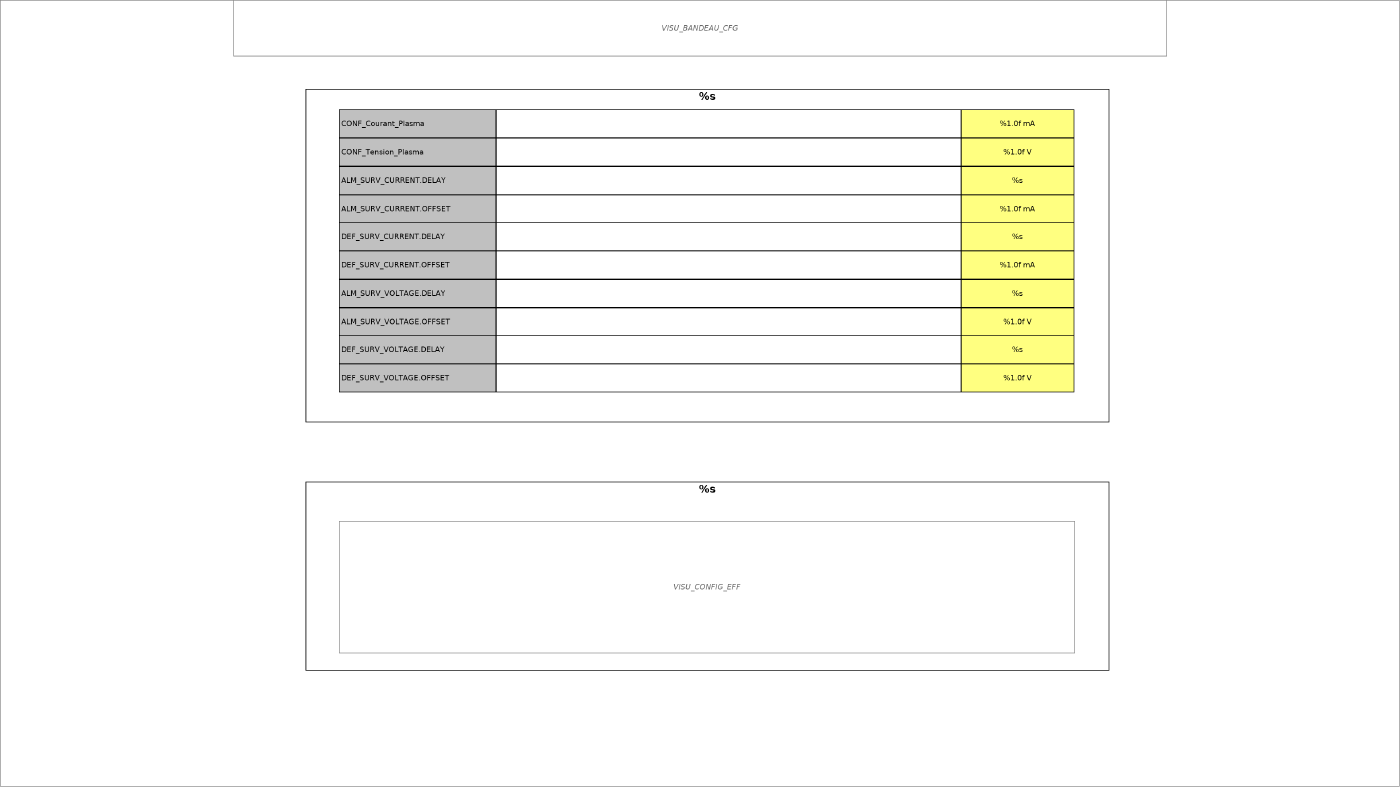
VISUALIZATION VISU_CONFIG_EFFLUV  // 1920x1080, background image fond_blanc_1280_1024
    Frame (320,0 1280x77)
        shows VISU_BANDEAU_CFG()
    RoundedRectangle (419,122 1102x457), "%s", text list: 'TextList_Config_EFFLUVAGE', text index: 0
    Rectangle (465,150 215x39), "CONF_Courant_Plasma"
    Rectangle (680,150 638x39), text list: 'TextList_Config_EFFLUVAGE', text index: 8
    Rectangle (1318,150 155x39), "%1.0f mA", text variable: PRG_EFFLUVAGE.Effluvage.ALEFF.CONF_Courant_Plasma, input disabled if: NOT Global_Variables.PRG_USER.ACTU_USER.CONF_MACHINE
        OnMouseClick: write the text variable via InputWithLimits, min 0, max 100
    Rectangle (465,189 215x39), "CONF_Tension_Plasma"
    Rectangle (680,189 638x39), text list: 'TextList_Config_EFFLUVAGE', text index: 9
    Rectangle (1318,189 155x39), "%1.0f V", text variable: PRG_EFFLUVAGE.Effluvage.ALEFF.CONF_Tension_Plasma, input disabled if: NOT Global_Variables.PRG_USER.ACTU_USER.CONF_MACHINE
        OnMouseClick: write the text variable via InputWithLimits, min 0, max 100
    Rectangle (465,228 215x39), "ALM_SURV_CURRENT.DELAY"
    Rectangle (680,228 638x39), text list: 'TextList_Config_EFFLUVAGE', text index: 11
    Rectangle (1318,228 155x39), "%s", text variable: PRG_EFFLUVAGE.Effluvage.ALEFF.ALM_Surv_Current.DELAY, input disabled if: NOT Global_Variables.PRG_USER.ACTU_USER.CONF_MACHINE
        OnMouseClick: write the text variable via InputWithLimits, min 0
    Rectangle (465,267 215x39), "ALM_SURV_CURRENT.OFFSET"
    Rectangle (680,267 638x39), text list: 'TextList_Config_EFFLUVAGE', text index: 12
    Rectangle (1318,267 155x39), "%1.0f mA", text variable: PRG_EFFLUVAGE.Effluvage.ALEFF.VAR_ALM_SURV_CURRENT.OFFSET, input disabled if: NOT Global_Variables.PRG_USER.ACTU_USER.CONF_MACHINE
        OnMouseClick: write the text variable via InputWithLimits, min 0, max 100
    Rectangle (465,305 215x39), "DEF_SURV_CURRENT.DELAY"
    Rectangle (680,305 638x39), text list: 'TextList_Config_EFFLUVAGE', text index: 13
    Rectangle (1318,305 155x39), "%s", text variable: PRG_EFFLUVAGE.Effluvage.ALEFF.DEF_Surv_Current.DELAY, input disabled if: NOT Global_Variables.PRG_USER.ACTU_USER.CONF_MACHINE
        OnMouseClick: write the text variable via InputWithLimits, min 0
    Rectangle (465,344 215x39), "DEF_SURV_CURRENT.OFFSET"
    Rectangle (680,344 638x39), text list: 'TextList_Config_EFFLUVAGE', text index: 14
    Rectangle (1318,344 155x39), "%1.0f mA", text variable: PRG_EFFLUVAGE.Effluvage.ALEFF.VAR_DEF_SURV_CURRENT.OFFSET, input disabled if: NOT Global_Variables.PRG_USER.ACTU_USER.CONF_MACHINE
        OnMouseClick: write the text variable via InputWithLimits, min 0, max 100
    RoundedRectangle (419,661 1102x259), "%s", text list: 'TextList_Config_EFFLUVAGE', text index: 0
    Frame (465,715 1009x181)
        shows VISU_CONFIG_EFF(m_Input_PRG_EFFLUVAGE := PRG_EFFLUVAGE)
    Rectangle (465,383 215x39), "ALM_SURV_VOLTAGE.DELAY"
    Rectangle (680,383 638x39), text list: 'TextList_Config_EFFLUVAGE', text index: 11
    Rectangle (1318,383 155x39), "%s", text variable: PRG_EFFLUVAGE.Effluvage.ALEFF.ALM_Surv_Voltage.DELAY, input disabled if: NOT Global_Variables.PRG_USER.ACTU_USER.CONF_MACHINE
        OnMouseClick: write the text variable via InputWithLimits, min 0
    Rectangle (465,422 215x39), "ALM_SURV_VOLTAGE.OFFSET"
    Rectangle (680,422 638x39), text list: 'TextList_Config_EFFLUVAGE', text index: 12
    Rectangle (1318,422 155x39), "%1.0f V", text variable: PRG_EFFLUVAGE.Effluvage.ALEFF.VAR_ALM_SURV_VOLTAGE.OFFSET, input disabled if: NOT Global_Variables.PRG_USER.ACTU_USER.CONF_MACHINE
        OnMouseClick: write the text variable via InputWithLimits, min 0, max 100
    Rectangle (465,460 215x39), "DEF_SURV_VOLTAGE.DELAY"
    Rectangle (680,460 638x39), text list: 'TextList_Config_EFFLUVAGE', text index: 13
    Rectangle (1318,460 155x39), "%s", text variable: PRG_EFFLUVAGE.Effluvage.ALEFF.DEF_Surv_Voltage.DELAY, input disabled if: NOT Global_Variables.PRG_USER.ACTU_USER.CONF_MACHINE
        OnMouseClick: write the text variable via InputWithLimits, min 0
    Rectangle (465,499 215x39), "DEF_SURV_VOLTAGE.OFFSET"
    Rectangle (680,499 638x39), text list: 'TextList_Config_EFFLUVAGE', text index: 14
    Rectangle (1318,499 155x39), "%1.0f V", text variable: PRG_EFFLUVAGE.Effluvage.ALEFF.VAR_DEF_SURV_VOLTAGE.OFFSET, input disabled if: NOT Global_Variables.PRG_USER.ACTU_USER.CONF_MACHINE
        OnMouseClick: write the text variable via InputWithLimits, min 0, max 100
END_VISUALIZATION

(* stored: Version 1.1.0.1, ProductVersion 3.1.4024.12
   Visu VISU_CONFIG_EFFLUV: Id {0cfb697d-746a-4c58-8203-a5824f4d87c4} *)
